FUNCTION_BLOCK FB_CTUD_ULINT (* counters (up-down-counter) *)
  (* Standard: 61131-3; Classification: standard counters; Description: Copyright (c) 2011 TU Wien ACIN This program and the accompanying materials are made available under the terms of the Eclipse Public License 2.0 which is available at https://www.eclipse.org/legal/epl-2.0/ SPDX-License-Identifier: EPL-2.0 *)
  (* Version 1.0, 2011-06-21, Monika Wenger, TU Wien ACIN *)
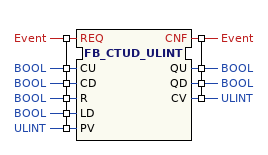
  EVENT_INPUT
    REQ WITH CD, PV, LD, CU, R; (* Service Request *)
  END_EVENT
  EVENT_OUTPUT
    CNF WITH QU, CV, QD; (* Confirmation of Requested Service *)
  END_EVENT
  VAR_INPUT
    CU : BOOL; (* Count up (Rising Edge Detection) *)
    CD : BOOL; (* Count down (Rising Edge Detection) *)
    R : BOOL; (* Reset *)
    LD : BOOL; (* Load *)
    PV : ULINT; (* Preset value *)
  END_VAR
  VAR_OUTPUT
    QU : BOOL; (* Output up count *)
    QD : BOOL; (* Output down count *)
    CV : ULINT; (* Count value *)
  END_VAR
  (* Service APPLICATION/RESOURCE: counters (up-down-counter) *)
END_FUNCTION_BLOCK
